PROGRAM OperatingModes
VAR
	aux:BOOL;
END_VAR

CASE GVL.Mode OF
	
	// Emergency stop
	Modes.STOP_EM:
		IF HMI.Bt_Rearm THEN
			gvl.Mode := modes.STOP_OP;
		END_IF
	
	// Operative stop
	Modes.STOP_OP:
		IF HMI.Bt_EmStop THEN
			GVL.Mode := Modes.STOP_EM;
		END_IF
		IF HMI.Bt_Run AND HMI.Sel_ManAuto THEN
			GVL.Mode := Modes.AUTO;
		END_IF
		IF NOT HMI.Sel_ManAuto THEN
			GVL.Mode := Modes.MAN;
		END_IF
		
	// Automatic
	Modes.AUTO:
		IF HMI.Bt_EmStop THEN
			GVL.Mode := Modes.STOP_EM;
		END_IF
		IF NOT HMI.Sel_ManAuto THEN
			GVL.Mode := Modes.MAN;
		END_IF
		IF HMI.Bt_Stop THEN
			GVL.Mode := Modes.STOP_OP;
		END_IF
		
	// Manual
	Modes.MAN:
		IF HMI.Bt_EmStop THEN
			GVL.Mode := Modes.STOP_EM;
		END_IF
		IF HMi.Sel_ManAuto THEN
			GVL.Mode := Modes.STOP_OP;
		END_IF
		
END_CASE

END_PROGRAM

(* stored: Version 1.1.0.1, ProductVersion 3.1.4024.9
   POU OperatingModes: Id {041e3654-c2e6-485e-9be9-b8cb759cbbc6}, SpecialFunc None *)
